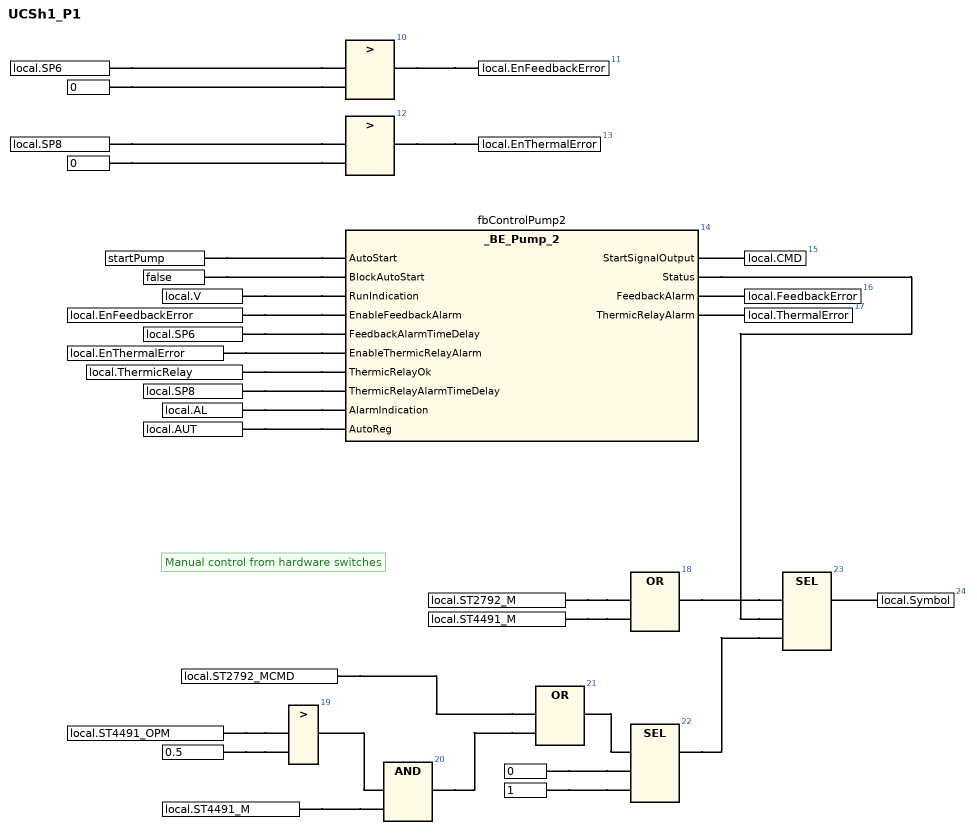
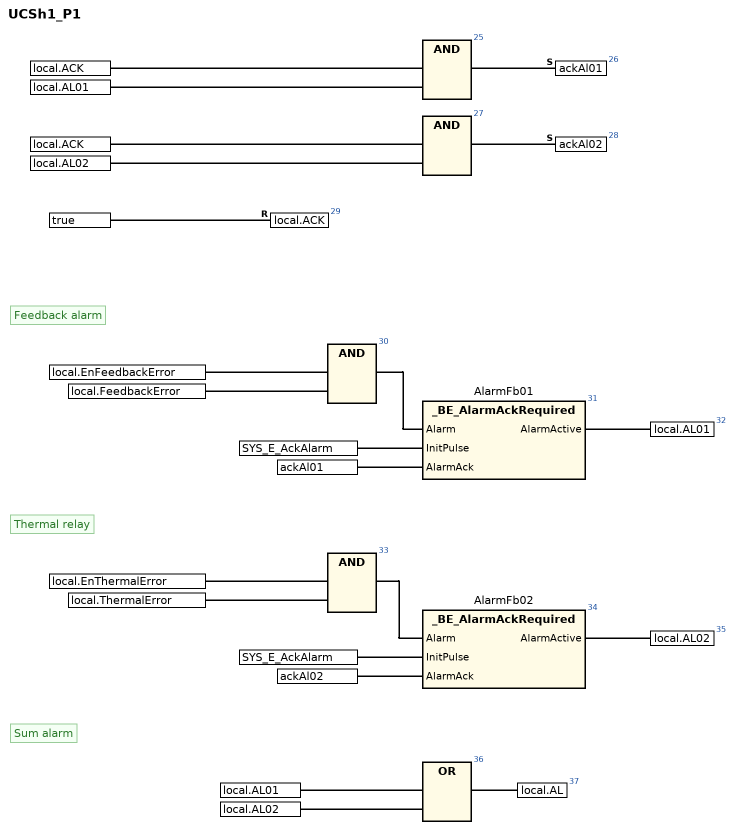
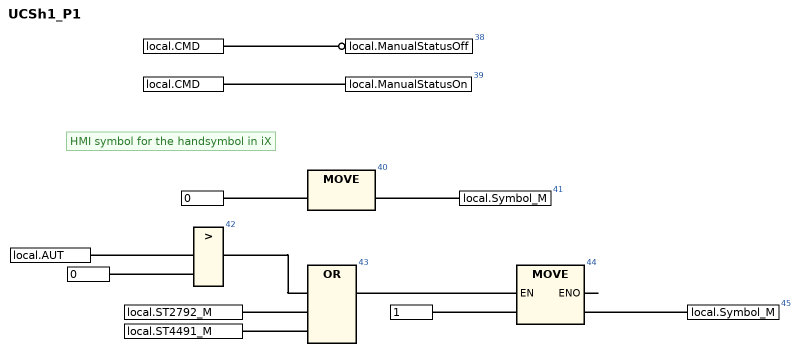
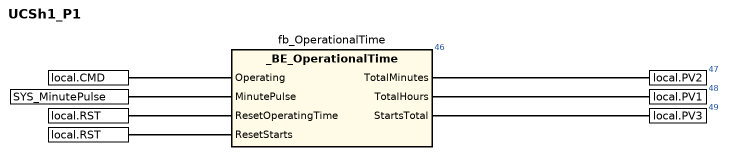
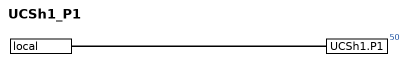
local := UCSh1.P1;
sv_op := UCSh1.SV1.OP;
fbExercise(
    EnableFunction := local.Ex_En,
    RunIndication := local.CMD,
    DaysBetweenExercise := local.SP4,
    HoursBetweenExercise := local.SP5,
    EnableDay := local.Ex_En_Day,
    ExerciseStartDay := local.SP9,
    EnableHourMinute := local.Ex_En_Time,
    ExerciseStartHour := local.SP10,
    ExerciseStartMinute := local.SP11,
    ExerciseRunTime := local.SP12,
    SecondPulse := SYS_SecondPulse,
    ClockArray := SYS_ArrayPlcTime,
    SecondsIncObjectOff := local.Ex_SecOff,
    SavedWorkingData := local.Ex_SavedData); // _BE_Exercise
local.V01 := fbExercise.ExerciseActive;
local.PV4 := fbExercise.DaysLeft;
local.PV5 := fbExercise.HoursLeft;
local.PV6 := fbExercise.MinutesLeft;
fbPumpStartCondition(
    CommandStart := local.V01,
    BlockStartSignalOutput := UCSh1.SWITCH = 0,
    EnableValveControl := true,
    ValveControlSignal := sv_op,
    ValueStartLimit := local.SP1,
    ValueStopLimit := local.SP2,
    EnableOutsideTempControl := local.EnTempControl,
    OutsideTemp := LB01.GT41.PV,
    OutsideTempDropsOrRise := FALSE,
    OutsideTempStartLimit := local.SP7,
    StopTimeDelay := local.SP3); // _BE_PumpStartConditions
startPump := fbPumpStartCondition.StartSignalOutput;
local.EnFeedbackError := local.SP6 > 0;
local.EnThermalError := local.SP8 > 0;
fbControlPump2(
    AutoStart := startPump,
    BlockAutoStart := false,
    RunIndication := local.V,
    EnableFeedbackAlarm := local.EnFeedbackError,
    FeedbackAlarmTimeDelay := local.SP6,
    EnableThermicRelayAlarm := local.EnThermalError,
    ThermicRelayOk := local.ThermicRelay,
    ThermicRelayAlarmTimeDelay := local.SP8,
    AlarmIndication := local.AL,
    AutoReg := local.AUT); // _BE_Pump_2
local.CMD := fbControlPump2.StartSignalOutput;
local.FeedbackError := fbControlPump2.FeedbackAlarm;
local.ThermalError := fbControlPump2.ThermicRelayAlarm;
// Manual control from hardware switches
local.Symbol := SEL(local.ST2792_M OR local.ST4491_M, fbControlPump2.Status, SEL(local.ST2792_MCMD OR local.ST4491_OPM > 0.5 AND local.ST4491_M, 0, 1));
ackAl01 S= local.ACK AND local.AL01;
ackAl02 S= local.ACK AND local.AL02;
local.ACK R= true;
// Feedback alarm
AlarmFb01(
    Alarm := local.EnFeedbackError AND local.FeedbackError,
    InitPulse := SYS_E_AckAlarm,
    AlarmAck := ackAl01); // _BE_AlarmAckRequired
local.AL01 := AlarmFb01.AlarmActive;
// Thermal relay
AlarmFb02(
    Alarm := local.EnThermalError AND local.ThermalError,
    InitPulse := SYS_E_AckAlarm,
    AlarmAck := ackAl02); // _BE_AlarmAckRequired
local.AL02 := AlarmFb02.AlarmActive;
// Sum alarm
local.AL := local.AL01 OR local.AL02;
local.ManualStatusOff := NOT local.CMD;
local.ManualStatusOn := local.CMD;
// HMI symbol for the handsymbol in iX
local.Symbol_M := 0;
IF local.AUT > 0 OR local.ST2792_M OR local.ST4491_M THEN _w1 := 1; END_IF
local.Symbol_M := _w1;
fb_OperationalTime(
    Operating := local.CMD,
    MinutePulse := SYS_MinutePulse,
    ResetOperatingTime := local.RST,
    ResetStarts := local.RST); // _BE_OperationalTime
local.PV2 := fb_OperationalTime.TotalMinutes;
local.PV1 := fb_OperationalTime.TotalHours;
local.PV3 := fb_OperationalTime.StartsTotal;
UCSh1.P1 := local;

END_PROGRAM

// Device/AREA1/B001/UC/Sh1/Sensor/GT1/UCSh1_GT1_Control
PROGRAM UCSh1_GT1_Control
VAR
	local:strSensor3_RegOutsideCompensation;
	gt_Min: TON;
	gt_Max: TON;
	reset_en: RS;
	FbRegulator: _BE_Regulator;
	cool_csp: REAL;
	cool_op: REAL;
	heatingOk: BOOL;
	fbOutsideComp: _BE_OutCompSevenSetPoint;
END_VAR
VAR // added by the converter: edge detectors and wires of the graphical bodies
    _w1, _w3, _w4 : ANY;
    _w2 : BOOL;
END_VAR

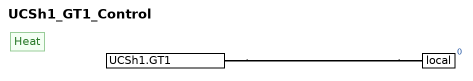
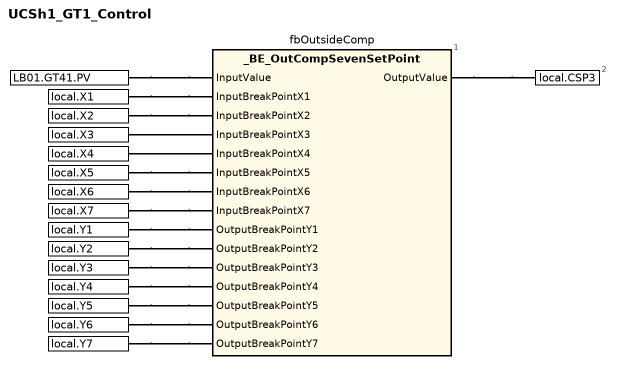
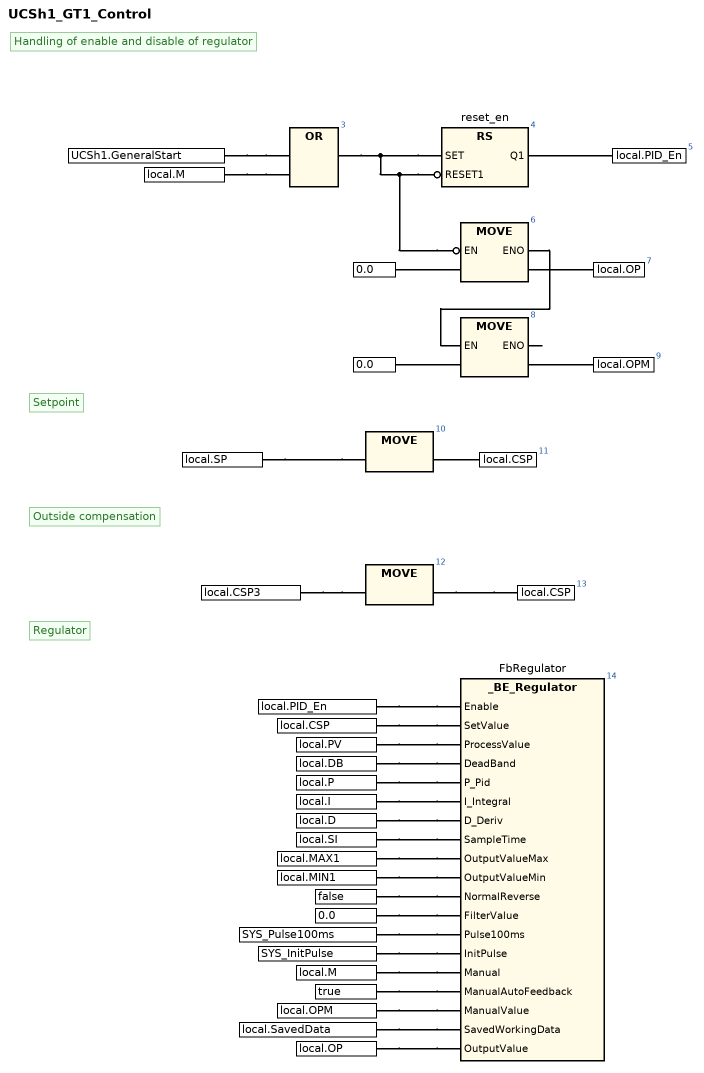
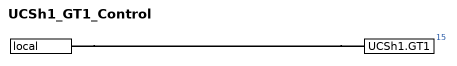
// Heat
local := UCSh1.GT1;
fbOutsideComp(
    InputValue := LB01.GT41.PV,
    InputBreakPointX1 := local.X1,
    InputBreakPointX2 := local.X2,
    InputBreakPointX3 := local.X3,
    InputBreakPointX4 := local.X4,
    InputBreakPointX5 := local.X5,
    InputBreakPointX6 := local.X6,
    InputBreakPointX7 := local.X7,
    OutputBreakPointY1 := local.Y1,
    OutputBreakPointY2 := local.Y2,
    OutputBreakPointY3 := local.Y3,
    OutputBreakPointY4 := local.Y4,
    OutputBreakPointY5 := local.Y5,
    OutputBreakPointY6 := local.Y6,
    OutputBreakPointY7 := local.Y7); // _BE_OutCompSevenSetPoint
local.CSP3 := fbOutsideComp.OutputValue;
// Handling of enable and disable of regulator
_w1 := UCSh1.GeneralStart OR local.M;
reset_en(SET := _w1, RESET1 := NOT _w1); // RS
local.PID_En := reset_en.Q1;
_w2 := NOT _w1;
IF _w2 THEN _w3 := 0.0; END_IF
local.OP := _w3;
IF _w2 THEN _w4 := 0.0; END_IF
local.OPM := _w4;
// Setpoint
local.CSP := local.SP;
// Outside compensation
local.CSP := local.CSP3;
// Regulator
FbRegulator(
    Enable := local.PID_En,
    SetValue := local.CSP,
    ProcessValue := local.PV,
    DeadBand := local.DB,
    P_Pid := local.P,
    I_Integral := local.I,
    D_Deriv := local.D,
    SampleTime := local.SI,
    OutputValueMax := local.MAX1,
    OutputValueMin := local.MIN1,
    NormalReverse := false,
    FilterValue := 0.0,
    Pulse100ms := SYS_Pulse100ms,
    InitPulse := SYS_InitPulse,
    Manual := local.M,
    ManualAutoFeedback := true,
    ManualValue := local.OPM,
    SavedWorkingData := local.SavedData,
    OutputValue := local.OP); // _BE_Regulator
UCSh1.GT1 := local;

END_PROGRAM

// Device/AREA1/B001/UC/Sh1/Sensor/GT1/UCSh1_GT1
PROGRAM UCSh1_GT1
VAR
	local:strSensor3_RegOutsideCompensation;
	gt_Min: TON;
	gt_Max: TON;
	ackFault: BOOL;
	ackLal: BOOL;
	ackHal: BOOL;
	AlarmAcknowledge01: _BE_AlarmAckRemote;
	AlarmAcknowledge02: _BE_AlarmAckRemote;
	AlarmAcknowledge03: _BE_AlarmAckRemote;
END_VAR
VAR // added by the converter: edge detectors and wires of the graphical bodies
    _w1, _w3, _w4 : ANY;
    _w2 : BOOL;
END_VAR

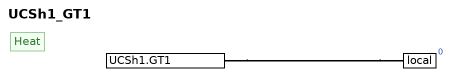
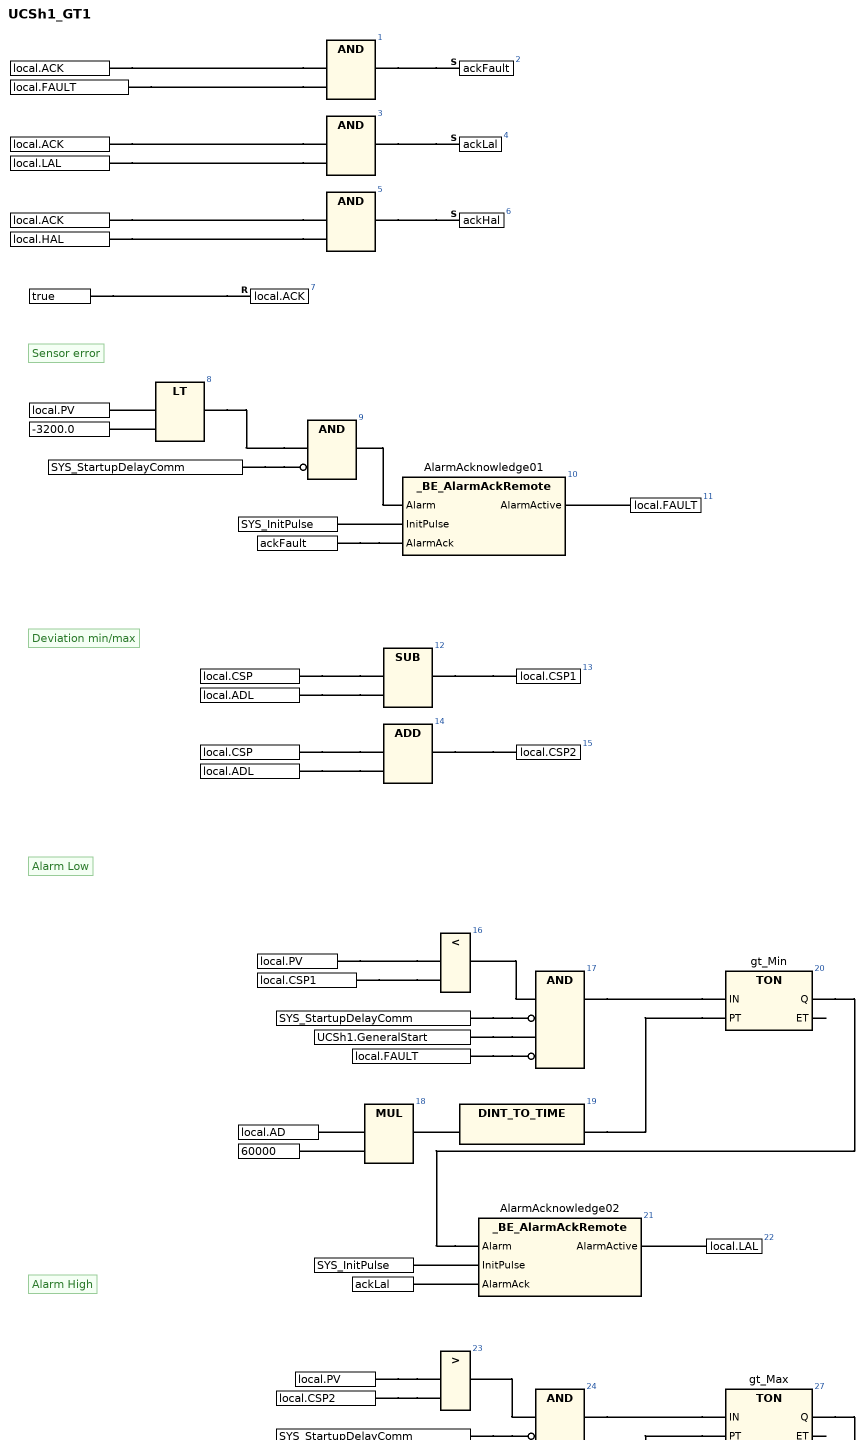
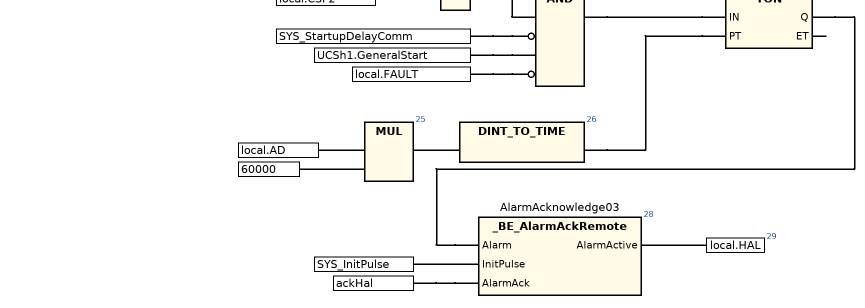
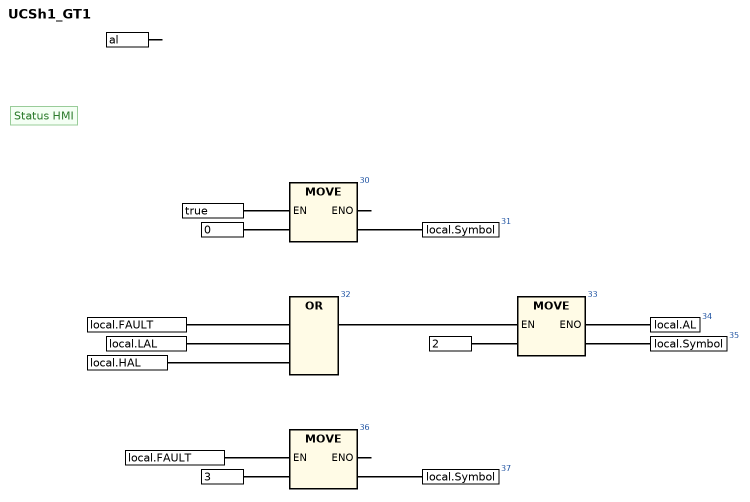
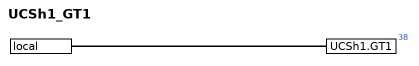
// Heat
local := UCSh1.GT1;
ackFault S= local.ACK AND local.FAULT;
ackLal S= local.ACK AND local.LAL;
ackHal S= local.ACK AND local.HAL;
local.ACK R= true;
// Sensor error
AlarmAcknowledge01(
    Alarm := local.PV < -3200.0 AND NOT SYS_StartupDelayComm,
    InitPulse := SYS_InitPulse,
    AlarmAck := ackFault); // _BE_AlarmAckRemote
local.FAULT := AlarmAcknowledge01.AlarmActive;
// Deviation min/max
local.CSP1 := local.CSP - local.ADL;
local.CSP2 := local.CSP + local.ADL;
// Alarm Low
gt_Min(IN := local.PV < local.CSP1 AND NOT SYS_StartupDelayComm AND UCSh1.GeneralStart AND NOT local.FAULT, PT := DINT_TO_TIME(local.AD * 60000)); // TON
AlarmAcknowledge02(Alarm := gt_Min.Q, InitPulse := SYS_InitPulse, AlarmAck := ackLal); // _BE_AlarmAckRemote
local.LAL := AlarmAcknowledge02.AlarmActive;
// Alarm High
gt_Max(IN := local.PV > local.CSP2 AND NOT SYS_StartupDelayComm AND UCSh1.GeneralStart AND NOT local.FAULT, PT := DINT_TO_TIME(local.AD * 60000)); // TON
AlarmAcknowledge03(Alarm := gt_Max.Q, InitPulse := SYS_InitPulse, AlarmAck := ackHal); // _BE_AlarmAckRemote
local.HAL := AlarmAcknowledge03.AlarmActive;
// Status HMI
IF true THEN _w1 := 0; END_IF
local.Symbol := _w1;
_w2 := local.FAULT OR local.LAL OR local.HAL;
IF _w2 THEN _w3 := 2; END_IF
local.AL := _w2;
local.Symbol := _w3;
IF local.FAULT THEN _w4 := 3; END_IF
local.Symbol := _w4;
UCSh1.GT1 := local;
// al: input not connected

END_PROGRAM

// Device/AREA1/B001/UC/Sh1/Sensor/GT2/UCSh1_GT2
PROGRAM UCSh1_GT2
VAR
	local:strSensor1;
	gt_Min: TON;
	gt_Max: TON;
	ackFault: BOOL;
	ackLal: BOOL;
	ackHal: BOOL;
	AlarmAcknowledge01: _BE_AlarmAckRemote;
	AlarmAcknowledge02: _BE_AlarmAckRemote;
	AlarmAcknowledge03: _BE_AlarmAckRemote;
END_VAR
VAR // added by the converter: edge detectors and wires of the graphical bodies
    _w1, _w3, _w4 : ANY;
    _w2 : BOOL;
END_VAR

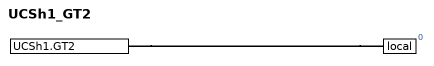
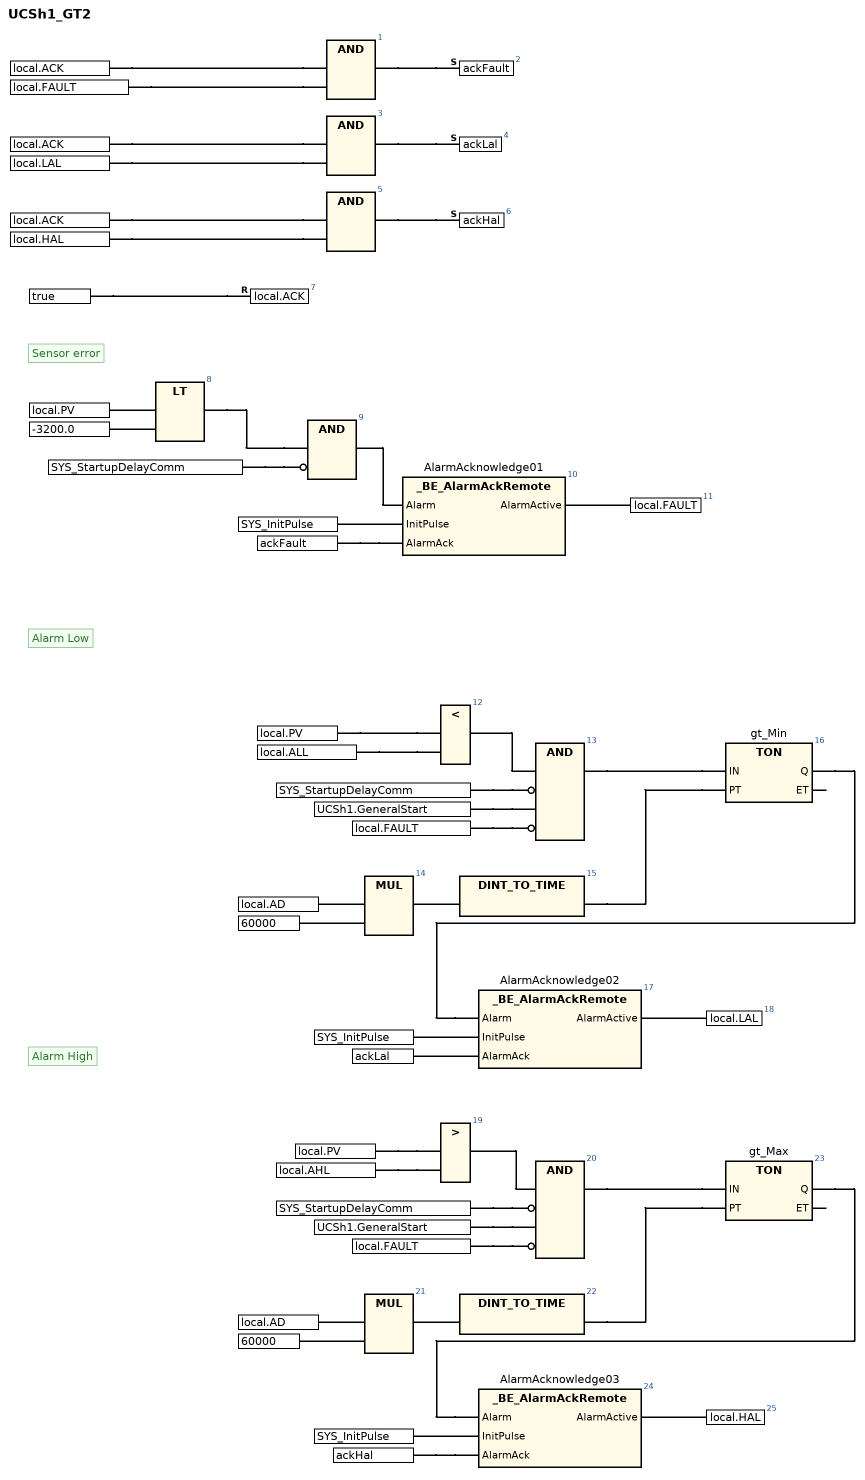
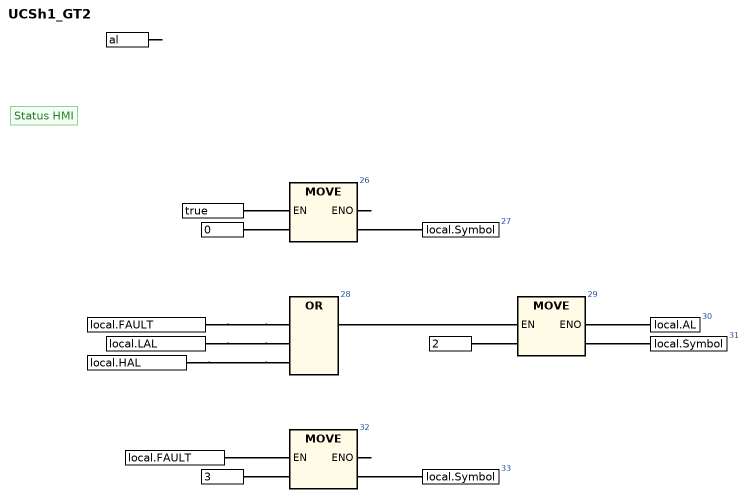
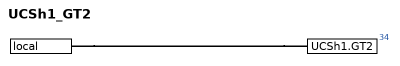
// note: 4 stored wires end on pins the file does not list and are not shown
local := UCSh1.GT2;
ackFault S= local.ACK AND local.FAULT;
ackLal S= local.ACK AND local.LAL;
ackHal S= local.ACK AND local.HAL;
local.ACK R= true;
// Sensor error
AlarmAcknowledge01(
    Alarm := local.PV < -3200.0 AND NOT SYS_StartupDelayComm,
    InitPulse := SYS_InitPulse,
    AlarmAck := ackFault); // _BE_AlarmAckRemote
local.FAULT := AlarmAcknowledge01.AlarmActive;
// Alarm Low
gt_Min(IN := local.PV < local.ALL AND NOT SYS_StartupDelayComm AND UCSh1.GeneralStart AND NOT local.FAULT, PT := DINT_TO_TIME(local.AD * 60000)); // TON
AlarmAcknowledge02(Alarm := gt_Min.Q, InitPulse := SYS_InitPulse, AlarmAck := ackLal); // _BE_AlarmAckRemote
local.LAL := AlarmAcknowledge02.AlarmActive;
// Alarm High
gt_Max(IN := local.PV > local.AHL AND NOT SYS_StartupDelayComm AND UCSh1.GeneralStart AND NOT local.FAULT, PT := DINT_TO_TIME(local.AD * 60000)); // TON
AlarmAcknowledge03(Alarm := gt_Max.Q, InitPulse := SYS_InitPulse, AlarmAck := ackHal); // _BE_AlarmAckRemote
local.HAL := AlarmAcknowledge03.AlarmActive;
// Status HMI
IF true THEN _w1 := 0; END_IF
local.Symbol := _w1;
_w2 := local.FAULT OR local.LAL OR local.HAL;
IF _w2 THEN _w3 := 2; END_IF
local.AL := _w2;
local.Symbol := _w3;
IF local.FAULT THEN _w4 := 3; END_IF
local.Symbol := _w4;
UCSh1.GT2 := local;
// al: input not connected

END_PROGRAM

// Device/AREA1/B001/UC/Sh1/Valve/UCSh1_SV1
PROGRAM UCSh1_SV1
VAR
	local:strValveExercise;
	FbAnalogueValve: _BE_AnalogueValve;
	fbExercise: _BE_Exercise;
	analogValue: REAL;
	valueFreezeProtection: REAL;
	FbAnalogOverride: _BE_AnalogueOverride;
	seqOutput: REAL;
END_VAR
VAR // added by the converter: edge detectors and wires of the graphical bodies
    _w1, _w2, _w3 : ANY;
END_VAR

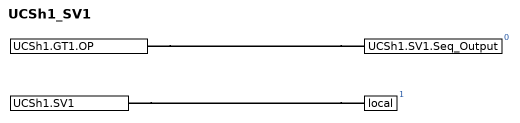
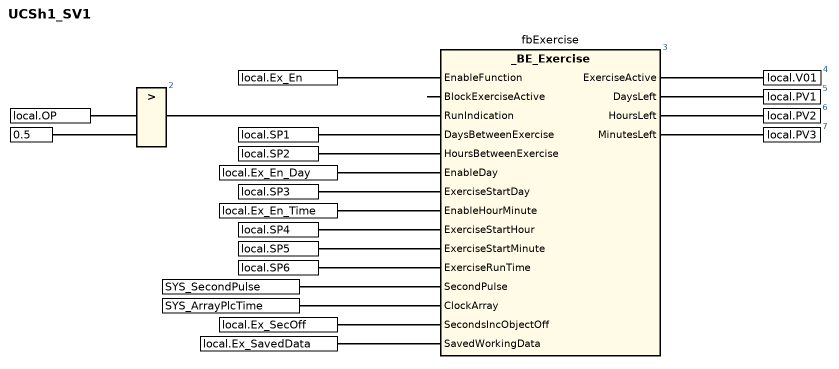
